FUNCTION_BLOCK FB_Co2MeanFlowCalculationHandler
VAR_INPUT
	serialCommData : ST_SerialCommReadData;
	flowControlParameters : ST_FlowControlParameters;
	startCalculation : BOOL;
END_VAR
VAR_OUTPUT
	meanReactorFlow : REAL;
END_VAR
VAR
	reactorFlow : REAL;
	flowMovingAvg : FB_MovingAverage;
	parameters : ST_FlowControlParameters;
	resetActive : BOOL;
END_VAR


reactorFlow := serialCommData.flowMeasurement;

// Calculate mean flow 
IF startCalculation THEN
	flowMovingAvg.startCalculation(
								start := TRUE,
								measurement := reactorFlow,
								windowS := flowControlParameters.movingAvgDurationSecs,
								intervalS := flowControlParameters.movingAvgShiftIntervalSecs,
								dtime := T#10MS,
								excludeUntilReady := flowControlParameters.excludeValuesPreFirstWindow);
	resetActive := FALSE;
ELSE
	IF NOT resetActive THEN
		flowMovingAvg.reset();
		resetActive := TRUE;
	END_IF
END_IF

meanReactorFlow := flowMovingAvg.value;

END_FUNCTION_BLOCK

(* stored: Version 1.1.0.1, ProductVersion 3.1.4024.9
   POU FB_Co2MeanFlowCalculationHandler: Id {9379d561-bf83-45df-82f1-1ed2e63f5583}, SpecialFunc None *)
